PROGRAM MAIN

VAR
	start : BOOL := FALSE;
	Tfill: TON;
	FILLING : BOOL := FALSE;
	WaterLevel : BOOL := FALSE;
	Level : REAL;
	Theat: TON;
    WaterTemp :REAL;
	HEATING : BOOL := FALSE;
	Tbrew: TON;
    WaterReady : BOOL := FALSE;
	BREWING : BOOL := FALSE;
    Tend: TON;
	
	CoffeeBrewed : BOOL := FALSE;
	Tready: TON;
	
	INTENSITY : INT;
	TIMER : TON;
	SugarLevel : INT :=1;
	SugarMessage : STRING(30);
	
	state : status := status.START;

	Tclean: TON;
END_VAR

CASE state OF

    status.START: 
        GVL.CoffeeReady := FALSE;
        FILLING := FALSE;
        HEATING := FALSE;
        BREWING := FALSE;
        WaterLevel := FALSE;
        WaterReady := FALSE;
		SugarMessage := '';
		IF start THEN
            state := status.LEVELCHECK;
        END_IF;       
		
	status.LEVELCHECK:
	IF Level >= 80 THEN
		state := status.HEAT;
		WaterLevel := TRUE;
	ELSIF Level < 80 THEN
 		state:=status.FILL;
	END_IF
	

    status.FILL:
		  Tfill(IN := TRUE, PT := T#8S);
		FILLING:= TRUE;
        FILLING := NOT WaterLevel; 
        WaterLevel := NOT FILLING;
        IF Tfill.Q THEN          
            Tfill(IN := FALSE);  
            FILLING := FALSE;    
            Level := 100;    
            State := status.HEAT;              
        END_IF
		IF NOT start THEN
			state := status.START;
		END_IF
		
	 status.HEAT:
        Theat (IN:=TRUE, PT := T#5S);
		HEATING := TRUE;
		HEATING := NOT WaterReady;
		WaterReady := NOT HEATING;
		IF Theat.Q THEN
			HEATING := FALSE;
			WaterTemp := 100;
			Level := Level - 10;
			Theat(IN:= FALSE);
			state := status.WATERREADY;
		END_IF
		
     status.WATERREADY:
	    WaterReady := TRUE;
        Theat(IN := TRUE, PT := T#5S);
        IF Theat.Q THEN
            WaterReady := FALSE;
            Theat(IN := FALSE);
			WaterTemp := 30;
            state := status.INTENS;
        END_IF

    status.INTENS:  
		 WaterLevel := FALSE;
         CASE INTENSITY OF
            1: Tbrew(IN := TRUE, PT := T#3S);
            2: Tbrew(IN := TRUE, PT := T#6S);
            3: Tbrew(IN := TRUE, PT := T#9S);
        ELSE
            Tbrew(IN := TRUE, PT := T#6S);  
        END_CASE

        BREWING := TRUE;  

        Tbrew (IN:=TRUE, PT:= T#5S);
        IF Tbrew.Q THEN
            BREWING := FALSE;     
            Tbrew(IN := FALSE); 
            State := status.SUGAR;  
            CoffeeBrewed := TRUE; 
        END_IF
    status.SUGAR: 
		IF CoffeeBrewed := TRUE THEN
		CASE SugarLevel OF
			1: SugarMessage := 'no sugar';
			2: SugarMessage := 'medium sugar';
			3: SugarMessage := 'full sugar';
		ELSE
            SugarMessage := 'invalid selection';
		END_CASE
		state := status.READY;
	END_IF
	
    status.READY:  
        Tready(IN := TRUE, PT := T#5S);
        IF Tready.Q THEN
            Tready(IN := FALSE);
            state := status.END;
            start := FALSE;
			GVL.CoffeeReady := TRUE;
			CoffeeBrewed := FALSE;
        END_IF
	
	status.END:  
        Tend(IN := TRUE, PT := T#5S);
        IF Tend.Q THEN
            Tend(IN := FALSE);
            state := status.CLEAN;
            start := FALSE;
			GVL.CoffeeReady := FALSE;
        END_IF;
		
	status.CLEAN:
	 IF GVL.CLEANING THEN
		 Tclean(IN:=TRUE, PT := T#5S);
		 IF Tclean.Q THEN
			 Tclean(IN:=FALSE);
			 state:=status.START;
		 END_IF
	ELSE state:=status.START;	 
	 END_IF
	 
	 

END_CASE;

END_PROGRAM

(* stored: Version 1.1.0.1, ProductVersion 3.1.4024.15
   POU MAIN: Id {de3beb21-c81c-41bb-870c-964d49ad45d1}, SpecialFunc None *)
